move 52,-178.7,1.9,2.8,8,-7.1;
move 52,-179.3,1.9,2.8,8.1,-7;
move 53,-179.9,1.9,2.8,8.1,-7;
move 54,-180.7,1.9,2.8,8.2,-6.9;
move 54,-181.5,1.8,2.8,8.2,-6.9;
move 55,-182.3,1.8,2.8,8.3,-6.8;
move 56,-183.3,1.8,2.8,8.3,-6.7;
move 56,-184.3,1.8,2.8,8.3,-6.7;
move 57,-185.4,1.7,2.8,8.4,-6.6;
move 57,-186.6,1.7,3.2,8.4,-6.5;
move 58,-187.8,1.6,3.2,8.5,-6.5;
move 59,-189,1.6,3.2,8.5,-6.4;
move 59,-190.2,1.5,3.2,8.5,-6.4;
move 59,-191.5,1.5,3.2,8.6,-6.3;
move 60,-192.8,1.4,3.2,8.6,-6.2;
move 60,-194.1,1.3,3.2,8.6,-6.2;
move 60,-195.4,1.3,3.2,8.7,-6.1;
move 60,-196.6,1.2,3.2,8.7,-6;
move 60,-197.8,1.1,3.2,8.7,-6;
move 59,-198.9,1,3.2,8.8,-5.9;
move 59,-199.9,1,3.2,8.8,-5.9;
move 59,-200.9,0.9,3.2,8.8,-5.8;
move 58,-201.8,0.8,3.2,8.9,-5.7;
move 57,-202.7,0.7,3.2,8.9,-5.7;
move 57,-203.5,0.7,2.8,8.9,-5.6;
move 56,-204.1,0.6,2.8,8.9,-5.5;
move 55,-204.8,0.5,2.8,9,-5.5;
move 55,-205.3,0.4,2.8,9,-5.4;
move 54,-205.8,0.3,2.8,9,-5.3;
move 53,-206.2,0.2,2.8,9,-5.3;
move 53,-206.5,0.1,2.8,9.1,-5.2;
move 52,-206.8,0.1,2.8,9.1,-5.1;
move 51,-207.1,-0,2.4,9.1,-5.1;
move 50,-207.2,-0.1,2.4,9.1,-5;
move 50,-207.3,-0.2,2.4,9.1,-4.9;
move 49,-207.4,-0.3,2.4,9.2,-4.9;
move 48,-207.5,-0.4,2.4,9.2,-4.8;
move 48,-207.5,-0.5,2.4,9.2,-4.7;
move 47,-207.4,-0.6,2.4,9.2,-4.7;
move 46,-207.3,-0.7,2.4,9.2,-4.6;
move 45,-207.2,-0.8,2,9.2,-4.5;
move 45,-207.1,-0.9,2,9.3,-4.5;
move 44,-206.9,-1,2,9.3,-4.4;
move 43,-206.7,-1.1,2,9.3,-4.3;
move 42,-206.6,-1.2,2,9.3,-4.3;
move 41,-206.4,-1.2,2,9.3,-4.2;
move 41,-206.2,-1.3,2,9.3,-4.1;
move 40,-206,-1.4,1.6,9.3,-4.1;
move 39,-205.8,-1.5,1.6,9.3,-4;
move 39,-205.6,-1.6,1.6,9.3,-3.9;
move 38,-205.4,-1.7,1.6,9.3,-3.9;
move 38,-205.3,-1.8,1.6,9.4,-3.8;
move 37,-205.1,-1.9,1.6,9.4,-3.7;
move 37,-205,-1.9,1.6,9.4,-3.7;
move 36,-204.8,-2,1.6,9.4,-3.6;
move 35,-204.7,-2.1,1.6,9.4,-3.5;
move 35,-204.6,-2.2,1.6,9.4,-3.4;
move 34,-204.5,-2.3,1.2,9.4,-3.4;
move 34,-204.4,-2.3,1.2,9.4,-3.3;
move 33,-204.3,-2.4,1.2,9.4,-3.2;
move 33,-204.2,-2.5,1.2,9.4,-3.2;
move 32,-204.2,-2.6,1.2,9.4,-3.1;
move 32,-204.1,-2.7,1.2,9.4,-3;
move 32,-204.1,-2.7,1.2,9.4,-3;
move 32,-204,-2.8,1.2,9.4,-2.9;
move 32,-204,-2.9,1.2,9.4,-2.8;
move 32,-204,-2.9,1.2,9.4,-2.8;
move 32,-204,-3,1.2,9.4,-2.7;
move 32,-204.1,-3,1.2,9.4,-2.6;
move 32,-204.1,-3.1,1.2,9.4,-2.6;
move 32,-204.2,-3.2,1.2,9.4,-2.5;
move 32,-204.2,-3.2,1.2,9.4,-2.4;
move 32,-204.3,-3.3,1.2,9.4,-2.4;
move 32,-204.4,-3.3,1.2,9.3,-2.3;
move 32,-204.6,-3.4,1.2,9.3,-2.2;
move 32,-204.7,-3.4,1.2,9.3,-2.2;
move 32,-204.9,-3.5,1.2,9.3,-2.1;
move 32,-205,-3.5,1.2,9.3,-2;
move 32,-205.2,-3.6,1.2,9.3,-2;
move 32,-205.4,-3.6,1.2,9.3,-1.9;
move 32,-205.7,-3.7,1.2,9.3,-1.9;
move 32,-205.9,-3.7,1.2,9.3,-1.8;
move 32,-206.2,-3.8,1.2,9.3,-1.7;
move 32,-206.5,-3.8,1.2,9.2,-1.7;
move 32,-206.8,-3.8,1.2,9.2,-1.6;
move 32,-207.1,-3.9,1.2,9.2,-1.6;
move 32,-207.4,-3.9,1.2,9.2,-1.5;
move 32,-207.7,-4,1.2,9.2,-1.5;
move 32,-208,-4,1.2,9.2,-1.4;
move 32,-208.3,-4.1,1.2,9.2,-1.4;
move 32,-208.6,-4.1,1.2,9.1,-1.3;
move 32,-208.9,-4.1,1.2,9.1,-1.3;
move 32,-209.2,-4.2,1.2,9.1,-1.2;
move 32,-209.4,-4.2,1.2,9.1,-1.2;
move 32,-209.7,-4.2,1.2,9.1,-1.1;
move 32,-209.9,-4.2,1.2,9.1,-1.1;
move 32,-210.2,-4.3,1.2,9,-1;
move 32,-210.4,-4.3,1.2,9,-1;
move 32,-210.5,-4.3,1.2,9,-1;
move 32,-210.7,-4.3,1.2,9,-0.9;
move 32,-210.9,-4.3,1.2,9,-0.9;
move 32,-211,-4.3,1.2,8.9,-0.9;
move 32,-211.1,-4.3,1.2,8.9,-0.8;
move 32,-211.2,-4.3,1.2,8.9,-0.8;
move 32,-211.3,-4.4,1.2,8.9,-0.8;
move 32,-211.4,-4.4,1.2,8.9,-0.7;
move 32,-211.5,-4.4,1.2,8.8,-0.7;
move 32,-211.5,-4.4,1.2,8.8,-0.7;
move 32,-211.6,-4.4,1.2,8.8,-0.6;
move 32,-211.7,-4.4,1.2,8.8,-0.6;




    ENDPROC

! function used to produce movement
    PROC move(num x, num z,num rx, num ry, num rz,num joint1)
     ConfJ\On;
     velocity := [300,1000,5000,1000];


     !!!! Method Two !!!!!!
     position :=RelTool(starting_position, x,0, z \Rx:=rx, \Ry:=ry, \Rz:=rz);
     joints := CalcJointT(position,Tooldata_9 \WObj:=Workobject_2);
     joints.robax.rax_1 :=joint1;
     MoveAbsJ joints,v800,z200,Tooldata_9,\WObj:=wobj0;
     !!!!!!!!!!!!!!!!!!!!!!!!!!!!!!

    ENDPROC



ENDMODULE
